(* IEC 61131-3 sources: controlforge-structured-text/manual-tests/formatting, 3 files *)

(* ---- expected-output.st ---- *)
(* Manual test: Code Formatting - Expected output *)
(* This file shows what unformatted-input.st should look like after formatting *)

// Test 1: Keyword casing (should become uppercase)
PROGRAM main
    VAR
        counter      : INT := 0;
        temperature  : REAL := 25.5;
        isRunning    : BOOL := TRUE;
        longVariableName : DINT := 100;
    END_VAR

    // Test 2: Indentation and operator spacing
    IF counter > 100 THEN
        counter := 0;
        temperature := temperature * 1.1;
    ELSIF counter > 50 THEN
        temperature := temperature * 0.99;
    ELSE
        temperature := temperature + 0.1;
    END_IF

    // Test 3: Nested blocks
    FOR i := 1 TO 10 BY 1 DO
        IF temperature > 50.0 THEN
            counter := counter + 1;
        END_IF
    END_FOR

    // Test 4: WHILE loop
    WHILE counter < 100 AND temperature < 80.0 DO
        counter := counter + 1;
    END_WHILE

    // Test 5: REPEAT..UNTIL
    REPEAT
        temperature := temperature - 0.1;
    UNTIL temperature <= 25.0
    END_REPEAT

    // Test 6: CASE statement
    CASE motorState OF
        STOPPED:
            message := 'Motor stopped';
        RUNNING:
            message := 'Motor running';
    ELSE
        message := 'Unknown state';
    END_CASE

    // Test 7: Comments should not be modified
    // this comment has if then else keywords
    (* block comment with var end_var inside *)

    // Test 8: Strings should not be modified
    message := 'Hello World';
    wideMsg := "Unicode Text";

END_PROGRAM

// Test 9: Function block with multiple VAR sections
FUNCTION_BLOCK fb_test
    VAR_INPUT
        start          : BOOL;
        speed_setpoint : REAL;
        enable         : BOOL := TRUE;
    END_VAR
    VAR_OUTPUT
        running      : BOOL;
        actual_speed : REAL;
    END_VAR
    VAR
        internal_state : INT;
        motor_on       : BOOL;
    END_VAR
    running := start AND enable;
END_FUNCTION_BLOCK

// Test 10: Function with return type
FUNCTION celsius_to_fahrenheit : REAL
    VAR_INPUT
        celsius : REAL;
    END_VAR
    celsius_to_fahrenheit := celsius * 9.0 / 5.0 + 32.0;
END_FUNCTION

(* ---- unformatted-input.st ---- *)
(* Manual test: Code Formatting - Unformatted input *)
(* Use Format Document to format this file and verify results *)
(* Linux: Ctrl+Shift+I  |  Windows/macOS: Shift+Alt+F  |  Any: Ctrl+Shift+P -> "Format Document" *)

// Test 1: Keyword casing (should become uppercase)
program main
var
counter:int:=0;
temperature:real:=25.5;
isRunning:bool:=true;
longVariableName:dint:=100;
end_var

// Test 2: Indentation and operator spacing
if counter>100 then
counter:=0;
temperature:=temperature*1.1;
elsif counter>50 then
temperature:=temperature*0.99;
else
temperature:=temperature+0.1;
end_if;

// Test 3: Nested blocks
for i:=1 to 10 by 1 do
if temperature>50.0 then
counter:=counter+1;
end_if;
end_for;

// Test 4: WHILE loop
while counter<100 and temperature<80.0 do
counter:=counter+1;
end_while;

// Test 5: REPEAT..UNTIL
repeat
temperature:=temperature-0.1;
until temperature<=25.0
end_repeat;

// Test 6: CASE statement
case motorState of
STOPPED:
message:='Motor stopped';
RUNNING:
message:='Motor running';
else
message:='Unknown state';
end_case;

// Test 7: Comments should not be modified
// this comment has if then else keywords
(* block comment with var end_var inside *)

// Test 8: Strings should not be modified
message:='Hello World';
wideMsg:="Unicode Text";

end_program

// Test 9: Function block with multiple VAR sections
function_block fb_test
var_input
start:bool;
speed_setpoint:real;
enable:bool:=true;
end_var
var_output
running:bool;
actual_speed:real;
end_var
var
internal_state:int;
motor_on:bool;
end_var
running:=start and enable;
end_function_block

// Test 10: Function with return type
function celsius_to_fahrenheit:real
var_input
celsius:real;
end_var
celsius_to_fahrenheit:=celsius*9.0/5.0+32.0;
end_function

(* ---- settings-variations.st ---- *)
(* Manual test: Formatting with different settings
   Test formatting behavior when VS Code settings are changed.
   After each setting change, format this file (Shift+Alt+F) and verify. *)

(* === Baseline: Default settings === *)
(* keywordCase: "upper", insertSpacesAroundOperators: true,
   alignVarDeclarations: true, trimTrailingWhitespace: true,
   insertFinalNewline: true *)

PROGRAM SettingsTest
VAR
    counter : INT := 0;
    temperature : REAL := 25.0;
    running : BOOL := TRUE;
    longName : DINT := 999;
END_VAR

counter := counter + 1;
temperature := temperature * 1.5 + 2.0;

IF running AND counter < 100 THEN
    running := FALSE;
END_IF

END_PROGRAM

(* === Test 1: keywordCase = "lower" === *)
(* Change setting: structured-text.format.keywordCase = "lower" *)
(* Format file, then verify: PROGRAM -> program, VAR -> var, etc. *)

(* === Test 2: keywordCase = "preserve" === *)
(* Change setting: structured-text.format.keywordCase = "preserve" *)
(* Manually type mixed case: Program, Var, If *)
(* Format file, verify: case is NOT changed *)

(* === Test 3: insertSpacesAroundOperators = false === *)
(* Change setting, format, verify: "counter:=counter+1" (no spaces) *)

(* === Test 4: alignVarDeclarations = false === *)
(* Change setting, format, verify: variable colons are NOT aligned *)

(* === Test 5: trimTrailingWhitespace = false === *)
(* Add trailing spaces to lines, format, verify: spaces preserved *)

(* === Test 6: insertFinalNewline = false === *)
(* Format, verify: no trailing newline at end of file *)

(* === Test 7: Format Selection (range formatting) === *)
(* Select only the IF block below, right-click > Format Selection *)
(* Verify: only selected range is formatted, rest unchanged *)
if running then
counter:=0;
end_if;

(* === Test 8: Idempotency === *)
(* Format this file, then format again immediately *)
(* Verify: second format produces no changes *)
